// TwinCAT 3 PLC project HOMS_Test_PLC
// ProgramVersion: 3.1.4020.5
// libraries:
//   Tc2_MC2, * (Beckhoff Automation GmbH)
//   Tc2_SerialCom, * (Beckhoff Automation GmbH)
//   Tc2_Standard, * (Beckhoff Automation GmbH)
//   Tc2_System, * (Beckhoff Automation GmbH)
//   Tc2_Utilities, * (Beckhoff Automation GmbH)
//   Tc3_Module, * (Beckhoff Automation GmbH)
//   VisuDialogs, * (System)
//   lcls-twincat-motion,0.0.0,SLAC
// project tree:
//   Common/POUs/Helpers/ FB_PI_E621_SerialDriver.TcPOU (not stored), FB_PI_E621_SerialTransaction.TcPOU (not stored)
//   DUTs/ DUT_MotionStage_Extras.TcDUT (not stored), ST_PiezoAxis.TcDUT (not stored), ST_RenishawEnc.TcDUT
//   / GlobalTextList.TcGTLO, PlcTask.TcTTO, Visualization Manager.TcVMO (not stored)
//   GVLs/ GVL_SerialIO.TcGVL (not stored)
//   POUs/ MAIN.TcPOU
//   POUs/Serial Comm/ PiezoSerial.TcPOU (not stored), P_Serial_Com.TcPOU (not stored)
//   VISUs/ Visualization.TcVIS, VISU_MotionStage.TcVIS
// real-time tasks:
//   TASK PlcTask: cycle T#10ms, priority 20, ADS port 350
//   TASK serial_com: cycle T#5ms, priority 5, ADS port 351
// motion (NC):
//   TASK NC-Task 1 SAF: cycle T#2ms, priority 4, ADS port 501
//   TASK NC-Task 1 SVB: cycle T#10ms, priority 8, ADS port 511
//   AXIS Axis_Yup (id 3)
//     Dynamic: Acceleration=0.2, Deceleration=0.2, DelayTime=0.008
//     Velo: Maximum=0.45
//     OtherSettings: AllowMotionCmdToSlave=true
//     encoder EncType=29
//       EncPara: ScaleFactorNumerator=1e-06, MaxCount=#xffffffff, ReferenceSystem=1
//         SoftEndMinControl: Enable=true, Range=6.2
//         SoftEndMaxControl: Enable=true, Range=16.3
//         Inc: RefSoftSyncMask=#x0000ffff
//     drive DrvType=24
//       DrvPara: Inverse=true
//         Analog: VeloReferenz=0.488275, ScaleFactorActTorque=0.1
//         TimeComp: TaskDelayCycles=1
//     controller CtrType=2
//       CtrPara: PriorControlFactor=1
//         PosDiffControl: Range=0.5
//         PID: PosKp=20, PosExtKp=5, DeadBandPosition=0.0004
//         Observer: BandWidth=20
//   AXIS Axis_Ydwn (id 4)
//     Dynamic: Acceleration=0.2, Deceleration=0.2, DelayTime=0.008
//     Velo: Maximum=0.45
//     OtherSettings: AllowMotionCmdToSlave=true
//     encoder EncType=29
//       EncPara: ScaleFactorNumerator=1e-06, MaxCount=#xffffffff, ReferenceSystem=1
//         SoftEndMinControl: Enable=true, Range=9.2
//         SoftEndMaxControl: Enable=true, Range=19.3
//         Inc: RefSoftSyncMask=#x0000ffff
//     drive DrvType=24
//       DrvPara: Inverse=true
//         Analog: VeloReferenz=0.488275, ScaleFactorActTorque=0.1
//         TimeComp: TaskDelayCycles=1
//     controller CtrType=2
//       CtrPara: PriorControlFactor=1
//         PosDiffControl: Range=0.5
//         PID: PosKp=20, PosExtKp=5, DeadBandPosition=0.0004
//         Observer: BandWidth=20
//   AXIS Axis_Xup (id 1)
//     Dynamic: Acceleration=2, Deceleration=2, DelayTime=0.008
//     Velo: Maximum=1
//     OtherSettings: AllowMotionCmdToSlave=true
//     encoder EncType=29
//       EncPara: ScaleFactorNumerator=1e-06, MaxCount=#xffffffff, ReferenceSystem=1
//         SoftEndMinControl: Enable=true, Range=22.7
//         SoftEndMaxControl: Enable=true, Range=24.9
//     drive DrvType=24
//       Analog: VeloReferenz=1.2206875, ScaleFactorActTorque=0.1
//       TimeComp: TaskDelayCycles=1
//     controller CtrType=2
//       CtrPara: PriorControlFactor=1
//         PosDiffControl: Range=0.1
//         PID: PosKp=10, PosExtKp=1, DeadBandPosition=0.0004
//         Observer: BandWidth=20
//   AXIS Axis_Xdwn (id 2)
//     Dynamic: Acceleration=2, Deceleration=2, DelayTime=0.008
//     Velo: Maximum=1
//     OtherSettings: AllowMotionCmdToSlave=true
//     encoder EncType=29
//       EncPara: ScaleFactorNumerator=1e-06, MaxCount=#xffffffff, ReferenceSystem=1
//         SoftEndMinControl: Enable=true, Range=23.5
//         SoftEndMaxControl: Enable=true, Range=25.7
//         Inc: RefSoftSyncMask=#x0000ffff
//     drive DrvType=24
//       DrvPara: Inverse=true
//         Analog: VeloReferenz=1.2206875, ScaleFactorActTorque=0.1
//         TimeComp: TaskDelayCycles=1
//     controller CtrType=2
//       CtrPara: PriorControlFactor=1
//         PosDiffControl: Range=0.1
//         PID: PosKp=10, PosExtKp=1, DeadBandPosition=0.0004
//         Observer: BandWidth=20
//   AXIS Axis_PitchCoarse (id 5)
//     General: UnitName=urad
//     Dynamic: Acceleration=390, Deceleration=390, DelayTime=0.008
//     Velo: Maximum=760
//     OtherSettings: AllowMotionCmdToSlave=true
//     encoder EncType=29
//       EncPara: ScaleFactorNumerator=0.001949317739, MaxCount=#xffffffff, ReferenceSystem=1
//         SoftEndMinControl: Enable=true, Range=16200
//         SoftEndMaxControl: Enable=true, Range=20600
//         Inc: RefSoftSyncMask=#x0000ffff
//     drive DrvType=24
//       Analog: VeloReferenz=761.4424951, ScaleFactorActTorque=0.1
//       TimeComp: TaskDelayCycles=1
//     controller CtrType=2
//       CtrPara: PriorControlFactor=1
//         PosDiffControl: Range=195
//         PID: PosExtKp=1, DeadBandPosition=0.5
//         Observer: BandWidth=20
//   AXIS Axis_Bender (id 6)
//     Dynamic: Acceleration=0.1, Deceleration=0.1, DelayTime=0.008
//     Velo: Maximum=0.19
//     OtherSettings: AllowMotionCmdToSlave=true
//     encoder EncType=29
//       EncPara: ScaleFactorNumerator=1e-06, Inverse=true, MaxCount=#xffffffff, ReferenceSystem=1
//         Inc: RefSoftSyncMask=#x0000ffff
//     drive DrvType=24
//       DrvPara: Inverse=true
//         Analog: VeloReferenz=0.19531, ScaleFactorActTorque=0.1
//         TimeComp: TaskDelayCycles=1
//     controller CtrType=2
//       CtrPara: PriorControlFactor=1
//         PosDiffControl: Range=0.0003
//         PID: PosKp=10, PosExtKp=1, DeadBandPosition=4e-05
//         Observer: BandWidth=20
// I/O:
//   DEVICE Device 3 (EtherCAT), AmsNetId 172.21.148.46.4.1
//     Term 1 (EK1100) [EK1100 EtherCAT Coupler (2A E-Bus)]
//       Term 2 (EL7041-1000) - Xup [EL7041-1000 1Ch. Stepper motor output stage (50V, 5A, standard)]
//       Term 3 (EL7041-1000) - Xdwn [EL7041-1000 1Ch. Stepper motor output stage (50V, 5A, standard)]
//       Term 4 (EL7041-1000) - Yup [EL7041-1000 1Ch. Stepper motor output stage (50V, 5A, standard)]
//       Term 5 (EL7041-1000) - Ydwn [EL7041-1000 1Ch. Stepper motor output stage (50V, 5A, standard)]
//       Term 6 (EL7041-1000) - PitchCourse [EL7041-1000 1Ch. Stepper motor output stage (50V, 5A, standard)]
//       Term 7 (EL7041-1000) - Bender [EL7041-1000 1Ch. Stepper motor output stage (50V, 5A, standard)]
//       Term 8 (EL6001) - PitchFine [EL6001 Interface (RS232)]
//       Term 9 (EL5042) - X [EL5042 2Ch. BiSS-C Encoder]
//       Term 10 (EL5042) - Y [EL5042 2Ch. BiSS-C Encoder]
//       Term 11 (EL5042) - PitchBender [EL5042 2Ch. BiSS-C Encoder]
//       Term 12 (EL1004) - STO [EL1004 4Ch. Dig. Input 24V, 3ms]
//       Term 13 (EL9505) - BenderLim [EL9505 Power supply terminal 5V]
//       Term 14 (EL9011) [EL9011 End Terminal]
// variable links:
//   (this object) <-> Device 3 (EtherCAT)/Term 1 (EK1100)/Term 10 (EL5042) - Y
//     Enc/Inputs/In/nComState @bit 1 <-> WcState/InputToggle
//     Enc/Inputs/In/nComState <-> WcState/WcState
//     Enc/Inputs/In/nDataIn1 <-> FB Inputs Channel 1/Position
//     Enc/Inputs/In/nDataIn1 <-> FB Inputs Channel 2/Position
//     Enc/Inputs/In/nState1 @bit 12 <-> FB Inputs Channel 1/Status/Diag
//     Enc/Inputs/In/nState1 @bit 12 <-> FB Inputs Channel 2/Status/Diag
//     Enc/Inputs/In/nState1 @bit 1 <-> FB Inputs Channel 1/Status/Error
//     Enc/Inputs/In/nState1 @bit 1 <-> FB Inputs Channel 2/Status/Error
//     Enc/Inputs/In/nState1 @bit 14 <-> FB Inputs Channel 1/Status/Input cycle counter
//     Enc/Inputs/In/nState1 @bit 14 <-> FB Inputs Channel 2/Status/Input cycle counter
//     Enc/Inputs/In/nState1 @bit 2 <-> FB Inputs Channel 1/Status/Ready
//     Enc/Inputs/In/nState1 @bit 2 <-> FB Inputs Channel 2/Status/Ready
//     Enc/Inputs/In/nState1 @bit 13 <-> FB Inputs Channel 1/Status/TxPDO State
//     Enc/Inputs/In/nState1 @bit 13 <-> FB Inputs Channel 2/Status/TxPDO State
//     Enc/Inputs/In/nState1 <-> FB Inputs Channel 1/Status/Warning
//     Enc/Inputs/In/nState1 <-> FB Inputs Channel 2/Status/Warning
//   (this object) <-> Device 3 (EtherCAT)/Term 1 (EK1100)/Term 4 (EL7041-1000) - Yup
//     Drive/Inputs/In/nState1 @bit 3 <-> STM Status/Status/Error
//     Drive/Inputs/In/nState1 @bit 5 <-> STM Status/Status/Moving negative
//     Drive/Inputs/In/nState1 @bit 4 <-> STM Status/Status/Moving positive
//     Drive/Inputs/In/nState1 @bit 1 <-> STM Status/Status/Ready
//     Drive/Inputs/In/nState1 <-> STM Status/Status/Ready to enable
//     Drive/Inputs/In/nState1 @bit 6 <-> STM Status/Status/Torque reduced
//     Drive/Inputs/In/nState1 @bit 2 <-> STM Status/Status/Warning
//     Drive/Inputs/In/nState2 @bit 3 <-> STM Status/Status/Digital input 1
//     Drive/Inputs/In/nState2 @bit 4 <-> STM Status/Status/Digital input 2
//     Drive/Inputs/In/nState2 @bit 5 <-> STM Status/Status/Sync error
//     Drive/Inputs/In/nState2 @bit 7 <-> STM Status/Status/TxPDO Toggle
//     Drive/Inputs/In/nState4 @bit 1 <-> WcState/InputToggle
//     Drive/Inputs/In/nState4 <-> WcState/WcState
//     Drive/Outputs/Out/nCtrl1 <-> STM Control/Control/Enable
//     Drive/Outputs/Out/nCtrl1 @bit 2 <-> STM Control/Control/Reduce torque
//     Drive/Outputs/Out/nCtrl1 @bit 1 <-> STM Control/Control/Reset
//     Drive/Outputs/Out/nDataOut2[0] <-> STM Velocity/Velocity
//   (this object) <-> Device 3 (EtherCAT)/Term 1 (EK1100)/Term 5 (EL7041-1000) - Ydwn
//     Drive/Inputs/In/nState1 @bit 3 <-> STM Status/Status/Error
//     Drive/Inputs/In/nState1 @bit 5 <-> STM Status/Status/Moving negative
//     Drive/Inputs/In/nState1 @bit 4 <-> STM Status/Status/Moving positive
//     Drive/Inputs/In/nState1 @bit 1 <-> STM Status/Status/Ready
//     Drive/Inputs/In/nState1 <-> STM Status/Status/Ready to enable
//     Drive/Inputs/In/nState1 @bit 6 <-> STM Status/Status/Torque reduced
//     Drive/Inputs/In/nState1 @bit 2 <-> STM Status/Status/Warning
//     Drive/Inputs/In/nState2 @bit 3 <-> STM Status/Status/Digital input 1
//     Drive/Inputs/In/nState2 @bit 4 <-> STM Status/Status/Digital input 2
//     Drive/Inputs/In/nState2 @bit 5 <-> STM Status/Status/Sync error
//     Drive/Inputs/In/nState2 @bit 7 <-> STM Status/Status/TxPDO Toggle
//     Drive/Inputs/In/nState4 @bit 1 <-> WcState/InputToggle
//     Drive/Inputs/In/nState4 <-> WcState/WcState
//     Drive/Outputs/Out/nCtrl1 <-> STM Control/Control/Enable
//     Drive/Outputs/Out/nCtrl1 @bit 2 <-> STM Control/Control/Reduce torque
//     Drive/Outputs/Out/nCtrl1 @bit 1 <-> STM Control/Control/Reset
//     Drive/Outputs/Out/nDataOut2[0] <-> STM Velocity/Velocity
//   (this object) <-> Device 3 (EtherCAT)/Term 1 (EK1100)/Term 2 (EL7041-1000) - Xup
//     Drive/Inputs/In/nState1 @bit 3 <-> STM Status/Status/Error
//     Drive/Inputs/In/nState1 @bit 5 <-> STM Status/Status/Moving negative
//     Drive/Inputs/In/nState1 @bit 4 <-> STM Status/Status/Moving positive
//     Drive/Inputs/In/nState1 @bit 1 <-> STM Status/Status/Ready
//     Drive/Inputs/In/nState1 <-> STM Status/Status/Ready to enable
//     Drive/Inputs/In/nState1 @bit 6 <-> STM Status/Status/Torque reduced
//     Drive/Inputs/In/nState1 @bit 2 <-> STM Status/Status/Warning
//     Drive/Inputs/In/nState2 @bit 3 <-> STM Status/Status/Digital input 1
//     Drive/Inputs/In/nState2 @bit 4 <-> STM Status/Status/Digital input 2
//     Drive/Inputs/In/nState2 @bit 5 <-> STM Status/Status/Sync error
//     Drive/Inputs/In/nState2 @bit 7 <-> STM Status/Status/TxPDO Toggle
//     Drive/Inputs/In/nState4 @bit 1 <-> WcState/InputToggle
//     Drive/Inputs/In/nState4 <-> WcState/WcState
//     Drive/Outputs/Out/nCtrl1 <-> STM Control/Control/Enable
//     Drive/Outputs/Out/nCtrl1 @bit 2 <-> STM Control/Control/Reduce torque
//     Drive/Outputs/Out/nCtrl1 @bit 1 <-> STM Control/Control/Reset
//     Drive/Outputs/Out/nDataOut2[0] <-> STM Velocity/Velocity
//   (this object) <-> Device 3 (EtherCAT)/Term 1 (EK1100)/Term 9 (EL5042) - X
//     Enc/Inputs/In/nComState @bit 1 <-> WcState/InputToggle
//     Enc/Inputs/In/nComState <-> WcState/WcState
//     Enc/Inputs/In/nDataIn1 <-> FB Inputs Channel 1/Position
//     Enc/Inputs/In/nDataIn1 <-> FB Inputs Channel 2/Position
//     Enc/Inputs/In/nState1 @bit 12 <-> FB Inputs Channel 1/Status/Diag
//     Enc/Inputs/In/nState1 @bit 12 <-> FB Inputs Channel 2/Status/Diag
//     Enc/Inputs/In/nState1 @bit 1 <-> FB Inputs Channel 1/Status/Error
//     Enc/Inputs/In/nState1 @bit 1 <-> FB Inputs Channel 2/Status/Error
//     Enc/Inputs/In/nState1 @bit 14 <-> FB Inputs Channel 1/Status/Input cycle counter
//     Enc/Inputs/In/nState1 @bit 14 <-> FB Inputs Channel 2/Status/Input cycle counter
//     Enc/Inputs/In/nState1 @bit 2 <-> FB Inputs Channel 1/Status/Ready
//     Enc/Inputs/In/nState1 @bit 2 <-> FB Inputs Channel 2/Status/Ready
//     Enc/Inputs/In/nState1 @bit 13 <-> FB Inputs Channel 1/Status/TxPDO State
//     Enc/Inputs/In/nState1 @bit 13 <-> FB Inputs Channel 2/Status/TxPDO State
//     Enc/Inputs/In/nState1 <-> FB Inputs Channel 1/Status/Warning
//     Enc/Inputs/In/nState1 <-> FB Inputs Channel 2/Status/Warning
//   (this object) <-> Device 3 (EtherCAT)/Term 1 (EK1100)/Term 3 (EL7041-1000) - Xdwn
//     Drive/Inputs/In/nState1 @bit 3 <-> STM Status/Status/Error
//     Drive/Inputs/In/nState1 @bit 5 <-> STM Status/Status/Moving negative
//     Drive/Inputs/In/nState1 @bit 4 <-> STM Status/Status/Moving positive
//     Drive/Inputs/In/nState1 @bit 1 <-> STM Status/Status/Ready
//     Drive/Inputs/In/nState1 <-> STM Status/Status/Ready to enable
//     Drive/Inputs/In/nState1 @bit 6 <-> STM Status/Status/Torque reduced
//     Drive/Inputs/In/nState1 @bit 2 <-> STM Status/Status/Warning
//     Drive/Inputs/In/nState2 @bit 3 <-> STM Status/Status/Digital input 1
//     Drive/Inputs/In/nState2 @bit 4 <-> STM Status/Status/Digital input 2
//     Drive/Inputs/In/nState2 @bit 5 <-> STM Status/Status/Sync error
//     Drive/Inputs/In/nState2 @bit 7 <-> STM Status/Status/TxPDO Toggle
//     Drive/Inputs/In/nState4 @bit 1 <-> WcState/InputToggle
//     Drive/Inputs/In/nState4 <-> WcState/WcState
//     Drive/Outputs/Out/nCtrl1 <-> STM Control/Control/Enable
//     Drive/Outputs/Out/nCtrl1 @bit 2 <-> STM Control/Control/Reduce torque
//     Drive/Outputs/Out/nCtrl1 @bit 1 <-> STM Control/Control/Reset
//     Drive/Outputs/Out/nDataOut2[0] <-> STM Velocity/Velocity
//   (this object) <-> Device 3 (EtherCAT)/Term 1 (EK1100)/Term 11 (EL5042) - PitchBender
//     Enc/Inputs/In/nComState @bit 1 <-> WcState/InputToggle
//     Enc/Inputs/In/nComState <-> WcState/WcState
//     Enc/Inputs/In/nDataIn1 <-> FB Inputs Channel 1/Position
//     Enc/Inputs/In/nDataIn1 <-> FB Inputs Channel 2/Position
//     Enc/Inputs/In/nState1 @bit 12 <-> FB Inputs Channel 1/Status/Diag
//     Enc/Inputs/In/nState1 @bit 12 <-> FB Inputs Channel 2/Status/Diag
//     Enc/Inputs/In/nState1 @bit 1 <-> FB Inputs Channel 1/Status/Error
//     Enc/Inputs/In/nState1 @bit 1 <-> FB Inputs Channel 2/Status/Error
//     Enc/Inputs/In/nState1 @bit 14 <-> FB Inputs Channel 1/Status/Input cycle counter
//     Enc/Inputs/In/nState1 @bit 14 <-> FB Inputs Channel 2/Status/Input cycle counter
//     Enc/Inputs/In/nState1 @bit 2 <-> FB Inputs Channel 1/Status/Ready
//     Enc/Inputs/In/nState1 @bit 2 <-> FB Inputs Channel 2/Status/Ready
//     Enc/Inputs/In/nState1 @bit 13 <-> FB Inputs Channel 1/Status/TxPDO State
//     Enc/Inputs/In/nState1 @bit 13 <-> FB Inputs Channel 2/Status/TxPDO State
//     Enc/Inputs/In/nState1 <-> FB Inputs Channel 1/Status/Warning
//     Enc/Inputs/In/nState1 <-> FB Inputs Channel 2/Status/Warning
//   (this object) <-> Device 3 (EtherCAT)/Term 1 (EK1100)/Term 6 (EL7041-1000) - PitchCourse
//     Drive/Inputs/In/nState1 @bit 3 <-> STM Status/Status/Error
//     Drive/Inputs/In/nState1 @bit 5 <-> STM Status/Status/Moving negative
//     Drive/Inputs/In/nState1 @bit 4 <-> STM Status/Status/Moving positive
//     Drive/Inputs/In/nState1 @bit 1 <-> STM Status/Status/Ready
//     Drive/Inputs/In/nState1 <-> STM Status/Status/Ready to enable
//     Drive/Inputs/In/nState1 @bit 6 <-> STM Status/Status/Torque reduced
//     Drive/Inputs/In/nState1 @bit 2 <-> STM Status/Status/Warning
//     Drive/Inputs/In/nState2 @bit 3 <-> STM Status/Status/Digital input 1
//     Drive/Inputs/In/nState2 @bit 4 <-> STM Status/Status/Digital input 2
//     Drive/Inputs/In/nState2 @bit 5 <-> STM Status/Status/Sync error
//     Drive/Inputs/In/nState2 @bit 7 <-> STM Status/Status/TxPDO Toggle
//     Drive/Inputs/In/nState4 @bit 1 <-> WcState/InputToggle
//     Drive/Inputs/In/nState4 <-> WcState/WcState
//     Drive/Outputs/Out/nCtrl1 <-> STM Control/Control/Enable
//     Drive/Outputs/Out/nCtrl1 @bit 2 <-> STM Control/Control/Reduce torque
//     Drive/Outputs/Out/nCtrl1 @bit 1 <-> STM Control/Control/Reset
//     Drive/Outputs/Out/nDataOut2[0] <-> STM Velocity/Velocity
//   (this object) <-> Device 3 (EtherCAT)/Term 1 (EK1100)/Term 7 (EL7041-1000) - Bender
//     Drive/Inputs/In/nState1 @bit 3 <-> STM Status/Status/Error
//     Drive/Inputs/In/nState1 @bit 5 <-> STM Status/Status/Moving negative
//     Drive/Inputs/In/nState1 @bit 4 <-> STM Status/Status/Moving positive
//     Drive/Inputs/In/nState1 @bit 1 <-> STM Status/Status/Ready
//     Drive/Inputs/In/nState1 <-> STM Status/Status/Ready to enable
//     Drive/Inputs/In/nState1 @bit 6 <-> STM Status/Status/Torque reduced
//     Drive/Inputs/In/nState1 @bit 2 <-> STM Status/Status/Warning
//     Drive/Inputs/In/nState2 @bit 3 <-> STM Status/Status/Digital input 1
//     Drive/Inputs/In/nState2 @bit 4 <-> STM Status/Status/Digital input 2
//     Drive/Inputs/In/nState2 @bit 5 <-> STM Status/Status/Sync error
//     Drive/Inputs/In/nState2 @bit 7 <-> STM Status/Status/TxPDO Toggle
//     Drive/Inputs/In/nState4 @bit 1 <-> WcState/InputToggle
//     Drive/Inputs/In/nState4 <-> WcState/WcState
//     Drive/Outputs/Out/nCtrl1 <-> STM Control/Control/Enable
//     Drive/Outputs/Out/nCtrl1 @bit 2 <-> STM Control/Control/Reduce torque
//     Drive/Outputs/Out/nCtrl1 @bit 1 <-> STM Control/Control/Reset
//     Drive/Outputs/Out/nDataOut2[0] <-> STM Velocity/Velocity
//   HOMS_Test_PLC Instance <-> Device 3 (EtherCAT)/Term 1 (EK1100)/Term 10 (EL5042) - Y
//     PlcTask Inputs/Main.y_dwn_enc/Count <-> FB Inputs Channel 2/Position
//     PlcTask Inputs/Main.y_up_enc/Count <-> FB Inputs Channel 1/Position
//   HOMS_Test_PLC Instance <-> Device 3 (EtherCAT)/Term 1 (EK1100)/Term 12 (EL1004) - STO
//     PlcTask Inputs/Main.bSTOEnable1 <-> Channel 1/Input
//     PlcTask Inputs/Main.bSTOEnable2 <-> Channel 2/Input
//   HOMS_Test_PLC Instance <-> Device 3 (EtherCAT)/Term 1 (EK1100)/Term 2 (EL7041-1000) - Xup
//     PlcTask Inputs/Main.M3.bLimitBackwardEnable <-> STM Status/Status/Digital input 2
//     PlcTask Inputs/Main.M3.bLimitForwardEnable <-> STM Status/Status/Digital input 1
//   HOMS_Test_PLC Instance <-> Device 3 (EtherCAT)/Term 1 (EK1100)/Term 3 (EL7041-1000) - Xdwn
//     PlcTask Inputs/Main.M4.bLimitBackwardEnable <-> STM Status/Status/Digital input 2
//     PlcTask Inputs/Main.M4.bLimitForwardEnable <-> STM Status/Status/Digital input 1
//   HOMS_Test_PLC Instance <-> Device 3 (EtherCAT)/Term 1 (EK1100)/Term 4 (EL7041-1000) - Yup
//     PlcTask Inputs/Main.M1.bLimitBackwardEnable <-> STM Status/Status/Digital input 2
//     PlcTask Inputs/Main.M1.bLimitForwardEnable <-> STM Status/Status/Digital input 1
//   HOMS_Test_PLC Instance <-> Device 3 (EtherCAT)/Term 1 (EK1100)/Term 5 (EL7041-1000) - Ydwn
//     PlcTask Inputs/Main.M2.bLimitBackwardEnable <-> STM Status/Status/Digital input 2
//     PlcTask Inputs/Main.M2.bLimitForwardEnable <-> STM Status/Status/Digital input 1
//   HOMS_Test_PLC Instance <-> Device 3 (EtherCAT)/Term 1 (EK1100)/Term 6 (EL7041-1000) - PitchCourse
//     PlcTask Inputs/Main.M5.bLimitBackwardEnable <-> STM Status/Status/Digital input 2
//     PlcTask Inputs/Main.M5.bLimitForwardEnable <-> STM Status/Status/Digital input 1
//   HOMS_Test_PLC Instance <-> Device 3 (EtherCAT)/Term 1 (EK1100)/Term 7 (EL7041-1000) - Bender
//     PlcTask Inputs/Main.M6.bLimitBackwardEnable <-> STM Status/Status/Digital input 2
//     PlcTask Inputs/Main.M6.bLimitForwardEnable <-> STM Status/Status/Digital input 1
//   HOMS_Test_PLC Instance <-> Device 3 (EtherCAT)/Term 1 (EK1100)/Term 9 (EL5042) - X
//     PlcTask Inputs/Main.x_dwn_enc/Count <-> FB Inputs Channel 2/Position
//     PlcTask Inputs/Main.x_up_enc/Count <-> FB Inputs Channel 1/Position
//   HOMS_Test_PLC Instance <-> NC-Task 1 SAF/Axes/Axis_Bender
//     PlcTask Inputs/Main.M6.Axis.NcToPlc <-> Outputs/ToPlc
//     PlcTask Outputs/Main.M6.Axis.PlcToNc <-> Inputs/FromPlc
//   HOMS_Test_PLC Instance <-> NC-Task 1 SAF/Axes/Axis_PitchCoarse
//     PlcTask Inputs/Main.M5.Axis.NcToPlc <-> Outputs/ToPlc
//     PlcTask Outputs/Main.M5.Axis.PlcToNc <-> Inputs/FromPlc
//   HOMS_Test_PLC Instance <-> NC-Task 1 SAF/Axes/Axis_Xdwn
//     PlcTask Inputs/Main.M4.Axis.NcToPlc <-> Outputs/ToPlc
//     PlcTask Outputs/Main.M4.Axis.PlcToNc <-> Inputs/FromPlc
//   HOMS_Test_PLC Instance <-> NC-Task 1 SAF/Axes/Axis_Xup
//     PlcTask Inputs/Main.M3.Axis.NcToPlc <-> Outputs/ToPlc
//     PlcTask Outputs/Main.M3.Axis.PlcToNc <-> Inputs/FromPlc
//   HOMS_Test_PLC Instance <-> NC-Task 1 SAF/Axes/Axis_Ydwn
//     PlcTask Inputs/Main.M2.Axis.NcToPlc <-> Outputs/ToPlc
//     PlcTask Outputs/Main.M2.Axis.PlcToNc <-> Inputs/FromPlc
//   HOMS_Test_PLC Instance <-> NC-Task 1 SAF/Axes/Axis_Yup
//     PlcTask Inputs/Main.M1.Axis.NcToPlc <-> Outputs/ToPlc
//     PlcTask Outputs/Main.M1.Axis.PlcToNc <-> Inputs/FromPlc

CONFIGURATION HOMS_Test_PLC
    RESOURCE PLC ON TwinCAT3
        TASK PlcTask(INTERVAL := T#10ms, PRIORITY := 20);
        PROGRAM Main WITH PlcTask : Main;
    END_RESOURCE
END_CONFIGURATION

// ---- DUTs/ST_RenishawEnc.TcDUT
TYPE ST_RenishawEnc :
STRUCT
	Count	:	ULINT;
	Status	:	BOOL;
	Ref		:	ULINT;
END_STRUCT
END_TYPE

// ---- POUs/MAIN.TcPOU
PROGRAM Main
VAR		
    M1: DUT_MotionStage:=(nCommand:=3); // Yup
	M2: DUT_MotionStage:=(nCommand:=3); // Ydwn
	M3: DUT_MotionStage:=(nCommand:=3); // Xup
	M4: DUT_MotionStage:=(nCommand:=3); // Xdwn
	M5: DUT_MotionStage:=(nCommand:=3); // PitchCoarse
	M6: DUT_MotionStage:=(nCommand:=3); // Bender

	fbMotionStage_x_up, fbMotionStage_x_dwn, fbMotionStage_y_up, fbMotionStage_y_dwn, fbMotionStage_pitch, fbMotionStage_bender : FB_MotionStage;

	stoEnable AT %I* : BOOL;
	x_up_enc  AT %I*: ST_RenishawAbsEnc;
	x_dwn_enc  AT %I*: ST_RenishawAbsEnc;
	y_up_enc  AT %I*: ST_RenishawAbsEnc;
	y_dwn_enc  AT %I*: ST_RenishawAbsEnc;

	// Auto coupling function block
	fbAutoCoupleX : FB_GantryAutoCoupling;
	fbAutoCoupleY : FB_GantryAutoCoupling;
	bExecuteCoupleX : BOOL;
	bExecuteCoupleY : BOOL;
	bExecuteDecoupleX : BOOL;
	bExecuteDecoupleY : BOOL;
	bGantryAlreadyCoupledX : BOOL;
	bGantryAlreadyCoupledY : BOOL;
	
	// Gantry variables
	nCurrGantryX : LINT;
	nCurrGantryY : LINT;
	nGantryTolX : LINT := 25000;
	nGantryTolY : LINT := 25000;
END_VAR

// M2L0
// Buttons to enable motors: write 0 to enable, 2 to disable
M1.nEnableMode; // Yup
M2.nEnableMode; // Ydwn
M3.nEnableMode; // Xup
M4.nEnableMode; // Xdwn
M5.nEnableMode; // PitchCoarse

// Encoder Reference Values: Taken from HOMS_FEE project
y_up_enc.Ref := 14897597;
y_dwn_enc.Ref := 14551600;
x_up_enc.Ref := 23972500;
x_dwn_enc.Ref := 24766500;

// Gantry Differences to monitor
nCurrGantryY := ((ULINT_TO_LINT(y_up_enc.Count) - ULINT_TO_LINT(y_up_enc.Ref)) - (ULINT_TO_LINT(y_dwn_enc.Count) - ULINT_TO_LINT(y_dwn_enc.Ref)));
nCurrGantryX := ((ULINT_TO_LINT(x_up_enc.Count) - ULINT_TO_LINT(x_up_enc.Ref)) - (ULINT_TO_LINT(x_dwn_enc.Count) - ULINT_TO_LINT(x_dwn_enc.Ref)));

// E-stop
M1.bHardwareEnable := stoEnable;
M2.bHardwareEnable := stoEnable;
M3.bHardwareEnable := stoEnable;
M4.bHardwareEnable := stoEnable;
M5.bHardwareEnable := stoEnable;
M6.bHardwareEnable := stoEnable;

// Start Autocoupling
fbAutoCoupleX(nGantryTol:=nGantryTolX, Master:=M3, MasterEnc:=x_up_enc, Slave:=M4,
	          SlaveEnc:=x_dwn_enc, bExecuteCouple:=bExecuteCoupleX,
              bExecuteDecouple:=bExecuteDecoupleX,
              bGantryAlreadyCoupled=>bGantryAlreadyCoupledX);

fbAutoCoupleY(nGantryTol:=nGantryTolY, Master:=M1, MasterEnc:=y_up_enc, Slave:=M2,
	          SlaveEnc:=y_dwn_enc, bExecuteCouple:=bExecuteCoupleY,
              bExecuteDecouple:=bExecuteDecoupleY,
			  bGantryAlreadyCoupled=>bGantryAlreadyCoupledY);

fbMotionStage_y_up  (stMotionStage:=M1);
fbMotionStage_y_dwn (stMotionStage:=M2);
fbMotionStage_x_up  (stMotionStage:=M3);
fbMotionStage_x_dwn (stMotionStage:=M4);
fbMotionStage_pitch (stMotionStage:=M5);
fbMotionStage_bender (stMotionStage:=M6);

END_PROGRAM

// ---- GlobalTextList.TcGTLO
TEXTLIST GlobalTextList
  386 = '%f'
  406 = '%X'
  398 = '+'
  392 = '-'
  402 = '0 = Default Acceleration'
  404 = '0 = Default Deceleration'
  401 = 'Acceleration: %f'
  25 = 'Already Coupled: %f'
  396 = 'Clear'
  390 = 'Control'
  30 = 'Couple Motors'
  383 = 'Couple Status: 0 = Decoupled, 1 = Coupled'
  27 = 'Couple Status: TRUE if coupled'
  408 = 'Current Gantry Difference (Axilon): %f'
  29 = 'Current Gantry Difference in nm'
  409 = 'Current Gantry Difference in um'
  28 = 'Current Gantry Difference: %f'
  387 = 'Current Position'
  403 = 'Deceleration: %f'
  39 = 'Decouple Motors'
  41 = 'Disable'
  42 = 'Enable'
  37 = 'Enable Mode: %f'
  382 = 'Enable Status: 0 = Enabled, 2 = Disabled'
  384 = 'Ensure motors are coupled before attempting motion!'
  407 = 'Error Code'
  405 = 'Error:'
  394 = 'GO'
  395 = 'GO to set position'
  388 = 'High Limit Hit Indicator'
  385 = 'Low Limit Hit Indicator'
  389 = 'Moving:'
  34 = 'Pitch - MASTER'
  31 = 'Press To Couple Motors'
  40 = 'Press To Decouple Motors for independent control'
  391 = 'Set Position'
  399 = 'Settings'
  26 = 'Status'
  393 = 'Step Size'
  397 = 'STOP'
  35 = 'Units: mm'
  36 = 'Units: urad'
  400 = 'Velocity: %f'
  38 = 'Write 0 to Enable, 2 to Disable'
  33 = 'Xdwn - SLAVE'
  32 = 'Xup - MASTER'
  24 = 'Ydwn - SLAVE'
  23 = 'Yup - MASTER'
END_TEXTLIST

// ---- VISUs/Visualization.TcVIS
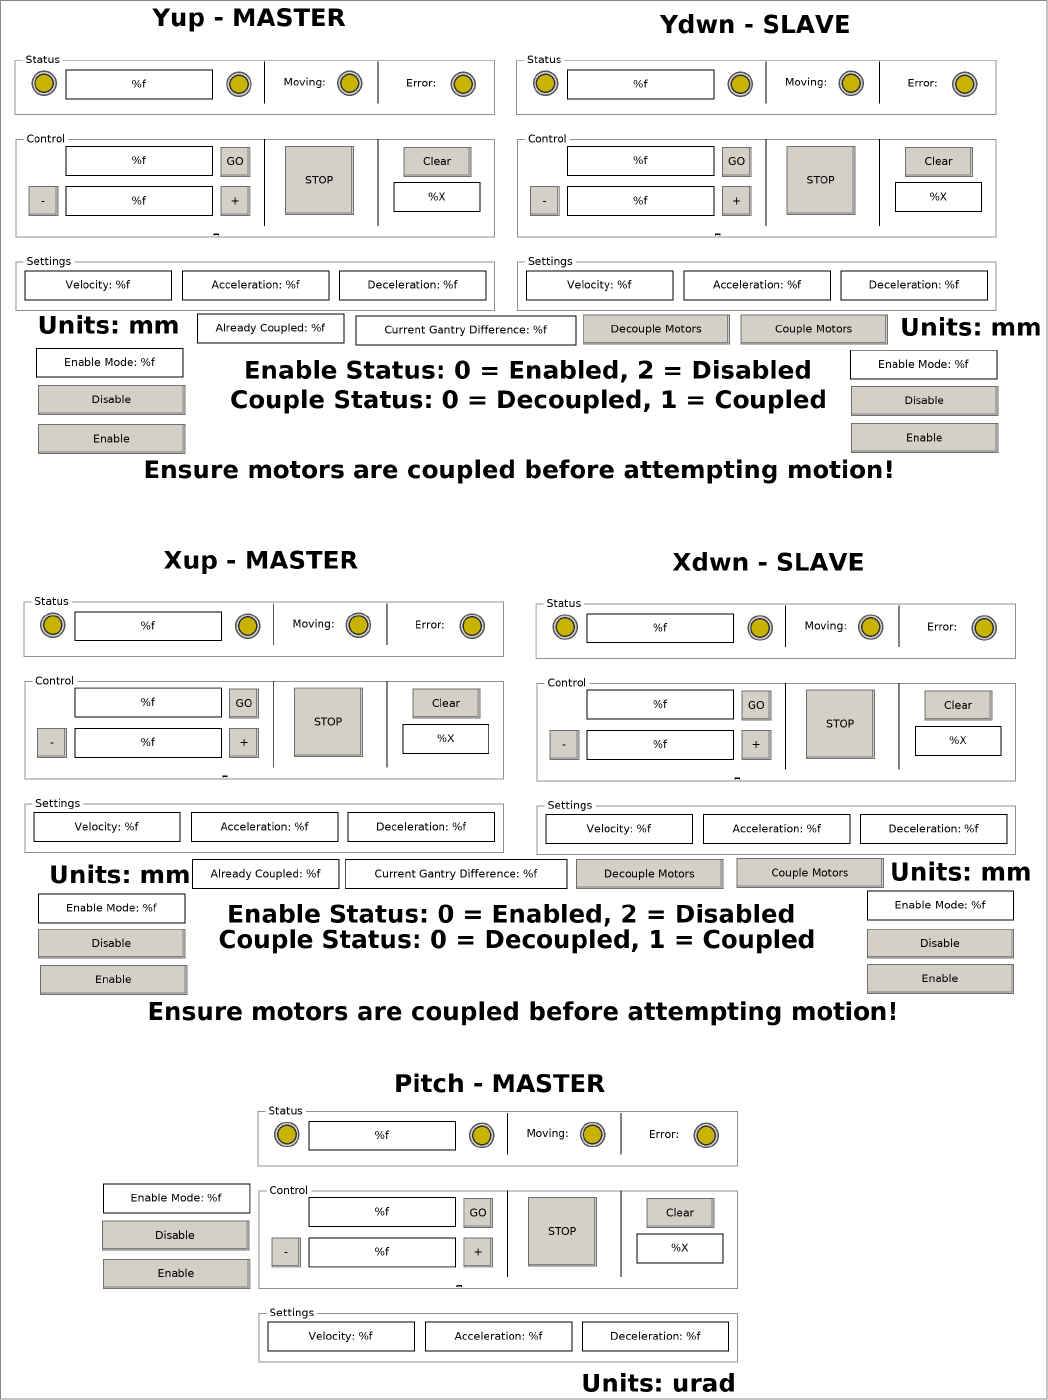
VISUALIZATION Visualization  // 1070x1429
    Label (14,2 481x31), "Yup - MASTER"
    Frame (0,36 520x300)
        shows VISU_MotionStage(VisuMotionStage := MAIN.M1, Extras := MAIN.M1_Extras)
    Frame (512,36 520x300)
        shows VISU_MotionStage(VisuMotionStage := MAIN.M2, Extras := MAIN.M2_Extras)
    Label (531,9 481x31), "Ydwn - SLAVE"
    Rectangle (201,320 150x30), "Already Coupled: %f", tooltip "Couple Status: TRUE if coupled", text variable: MAIN.bGantryAlreadyCoupledY
    Rectangle (363,322 225x30), "Current Gantry Difference: %f", tooltip "Current Gantry Difference in nm", text variable: MAIN.nCurrGantryY
    Button (756,321 150x30), "Couple Motors", tooltip "Press To Couple Motors", text variable: MAIN.bExecuteCoupleY
        OnMouseDown: execute { MAIN.bExecuteCoupleY := TRUE; }
    Frame (9,589 520x300)
        shows VISU_MotionStage(VisuMotionStage := MAIN.M3, Extras := MAIN.M3_Extras)
    Label (26,556 481x31), "Xup - MASTER"
    Frame (532,591 520x300)
        shows VISU_MotionStage(VisuMotionStage := MAIN.M4, Extras := MAIN.M4_Extras)
    Label (544,558 481x31), "Xdwn - SLAVE"
    Rectangle (196,877 150x30), "Already Coupled: %f", tooltip "Couple Status: TRUE if coupled", text variable: MAIN.bGantryAlreadyCoupledX
    Rectangle (352,877 227x30), "Current Gantry Difference: %f", tooltip "Current Gantry Difference in nm", text variable: MAIN.nCurrGantryX
    Frame (248,1109 520x300)
        shows VISU_MotionStage(VisuMotionStage := MAIN.M5, Extras := MAIN.M5_Extras)
    Label (270,1090 481x31), "Pitch - MASTER"
    Label (31,316 160x31), "Units: mm"
    Label (916,318 151x31), "Units: mm"
    Label (27,877 191x31), "Units: mm"
    Label (894,874 174x31), "Units: mm"
    Label (595,1396 155x31), "Units: urad"
    Rectangle (37,355 150x30), "Enable Mode: %f", tooltip "Write 0 to Enable, 2 to Disable", text variable: MAIN.M1.nEnableMode
    Rectangle (868,357 150x30), "Enable Mode: %f", tooltip "Write 0 to Enable, 2 to Disable", text variable: MAIN.M2.nEnableMode
    Button (595,321 150x30), "Decouple Motors", tooltip "Press To Decouple Motors for independent control"
        OnMouseDown: execute { MAIN.bExecuteDecoupleY := TRUE; }
    Button (39,393 150x30), "Disable"
        OnMouseDown: execute { MAIN.M1.nEnableMode := 2; }
    Button (39,433 150x30), "Enable", colour toggle: MAIN.bExecuteDecoupleY
        OnMouseDown: execute { MAIN.M1.nEnableMode := 0; }
    Button (869,394 150x30), "Disable"
        OnMouseDown: execute { MAIN.M2.nEnableMode := 2; }
    Button (869,432 150x30), "Enable", colour toggle: MAIN.bExecuteDecoupleY
        OnMouseDown: execute { MAIN.M2.nEnableMode := 0; }
    Button (588,877 150x30), "Decouple Motors", tooltip "Press To Decouple Motors for independent control"
        OnMouseDown: execute { MAIN.bExecuteDecoupleX := TRUE; }
    Button (752,876 150x30), "Couple Motors", tooltip "Press To Couple Motors", text variable: MAIN.bExecuteCoupleY
        OnMouseDown: execute { MAIN.bExecuteCoupleX := TRUE; }
    Rectangle (39,912 150x30), "Enable Mode: %f", tooltip "Write 0 to Enable, 2 to Disable", text variable: MAIN.M3.nEnableMode
    Button (39,948 150x30), "Disable"
        OnMouseDown: execute { MAIN.M3.nEnableMode := 2; }
    Button (41,985 150x30), "Enable", colour toggle: MAIN.bExecuteDecoupleY
        OnMouseDown: execute { MAIN.M3.nEnableMode := 0; }
    Rectangle (885,909 150x30), "Enable Mode: %f", tooltip "Write 0 to Enable, 2 to Disable", text variable: MAIN.M4.nEnableMode
    Button (885,948 150x30), "Disable"
        OnMouseDown: execute { MAIN.M4.nEnableMode := 2; }
    Button (885,984 150x30), "Enable", colour toggle: MAIN.bExecuteDecoupleY
        OnMouseDown: execute { MAIN.M4.nEnableMode := 0; }
    Rectangle (105,1208 150x30), "Enable Mode: %f", tooltip "Write 0 to Enable, 2 to Disable", text variable: MAIN.M5.nEnableMode
    Button (104,1246 150x30), "Disable"
        OnMouseDown: execute { MAIN.M5.nEnableMode := 2; }
    Button (105,1285 150x30), "Enable", colour toggle: MAIN.bExecuteDecoupleY
        OnMouseDown: execute { MAIN.M5.nEnableMode := 0; }
    Label (255,362 568x31), "Enable Status: 0 = Enabled, 2 = Disabled"
    Label (247,392 586x31), "Couple Status: 0 = Decoupled, 1 = Coupled"
    Label (238,917 568x31), "Enable Status: 0 = Enabled, 2 = Disabled"
    Label (235,943 586x31), "Couple Status: 0 = Decoupled, 1 = Coupled"
    Label (150,464 760x30), "Ensure motors are coupled before attempting motion!"
    Label (154,1017 760x30), "Ensure motors are coupled before attempting motion!"
END_VISUALIZATION

// ---- VISUs/VISU_MotionStage.TcVIS
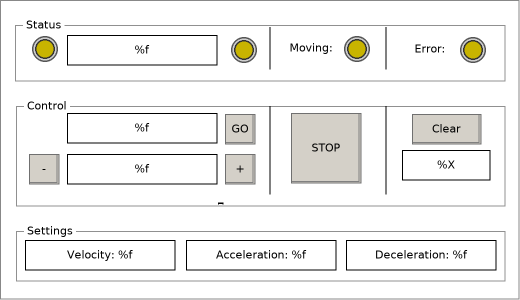
VISUALIZATION VISU_MotionStage  // 520x300
VAR_IN_OUT
	VisuMotionStage: DUT_MotionStage;
	Extras: DUT_MotionStage_Extras;
END_VAR
    GroupBox (15,17 490x64), "Status"
        Lamp1 (15,17 30x30), tooltip "Low Limit Hit Indicator", variable: Extras.bVisuLowLim, style: Lamp-Lamp1-Yellow
        Rectangle (52,18 150x30), "%f", tooltip "Current Position", text variable: VisuMotionStage.stAxisStatus.fActPosition
        Lamp1 (214,18 30x30), tooltip "High Limit Hit Indicator", variable: Extras.bVisuHighLim, style: Lamp-Lamp1-Yellow
        Lamp1 (327,17 30x30), variable: VisuMotionStage.bBusy, style: Lamp-Lamp1-Yellow
        Label (262,16 68x30), "Moving:"
        Line (371,52) (371,10)
        Lamp1 (443,18 30x30), variable: VisuMotionStage.bError, style: Lamp-Lamp1-Yellow
    Rectangle (218,203 5x0)
    GroupBox (16,98 489x108), "Control"
        Rectangle (51,15 150x30), "%f", tooltip "Set Position", text variable: VisuMotionStage.fPosition
            OnMouseDown: write the text variable via Default
        Button (13,56 30x30), "-"
            OnMouseDown: execute {
                VisuMotionStage.nCommand := 3;
                VisuMotionStage.fPosition := VisuMotionStage.stAxisStatus.fActPosition - Extras.fVisuStep;
                VisuMotionStage.bExecute := TRUE;
            }
        Rectangle (51,56 150x30), "%f", tooltip "Step Size", text variable: Extras.fVisuStep
            OnMouseDown: write the text variable via Default
        Button (209,16 30x30), "GO", tooltip "GO to set position"
            OnMouseDown: execute { VisuMotionStage.nCommand := 3; VisuMotionStage.bExecute := TRUE; }
        Line (254,96) (254,8)
        Line (370,96) (370,8)
        Button (396,16 69x30), "Clear"
            tap VisuMotionStage.bReset
        Button (275,15 70x70), "STOP", tooltip "GO to set position"
            OnMouseDown: execute { VisuMotionStage.bExecute := FALSE; }
        Button (209,56 30x30), "+"
            OnMouseDown: execute {
                VisuMotionStage.nCommand := 3;
                VisuMotionStage.fPosition := VisuMotionStage.stAxisStatus.fActPosition + Extras.fVisuStep;
                VisuMotionStage.bExecute := TRUE;
            }
    GroupBox (16,223 489x58), "Settings"
        Rectangle (9,17 150x30), "Velocity: %f", text variable: VisuMotionStage.fVelocity
            OnMouseDown: write the text variable via Default
        Rectangle (170,17 150x30), "Acceleration: %f", tooltip "0 = Default Acceleration", text variable: VisuMotionStage.fAcceleration
            OnMouseDown: write the text variable via Default
        Rectangle (330,17 150x30), "Deceleration: %f", tooltip "0 = Default Deceleration", text variable: VisuMotionStage.fDeceleration
            OnMouseDown: write the text variable via Default
    Line (270,69) (270,27)
    Label (396,34 68x30), "Error:"
    Rectangle (402,150 88x30), "%X", tooltip "Error Code", text variable: VisuMotionStage.stAxisStatus.nErrorId
END_VISUALIZATION
